ABB RobotStudio station: Simuleringsopgave_2_20200505-175028.rsstn

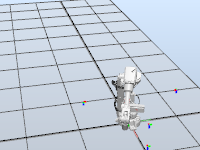
Station Simuleringsopgave_2 (saved by RobotStudio 7.0.8746.631)
Controller IRB_2600_20kg_1.65m_1
  mechanical unit ROB_1: IRB2600_20_165__02, 6 joints, base frame (0, 0, 0) mm
Layout (positions relative to the parent item):
  - IRB2600_20_165__02 [mechanism, from Robots\IRB2600_20_165_G_02.rslib] at (0, 0, 0) mm; joint values [-0.4129, 0.1779, 0.5307, -6.2924, 0.8625, 6.3308] (rad or m)
  - MyNewTool [mechanism] at (872.04, -382.72, 618.96) mm, rotated rx -179.6 ry 0 rz 153.96 deg
      TCP MyNewTool at (0, 0, 30) mm
      links: SimpleGripper
Attachment: MyNewTool is attached to IRB2600_20_165__02 / Link6
Targets, tools, work objects and paths stored in the station, written as RAPID:
! task T_ROB1
MODULE CalibData
  TASK PERS wobjdata Workobject_1:=[FALSE,TRUE,"",[[0,0,0],[1,0,0,0]],[[0,0,0],[1,0,0,0]]];
  PERS tooldata MyNewTool:=[TRUE,[[0,0,30],[1,0,0,0]],[1,[0,0,1],[1,0,0,0],0,0,0]];
ENDMODULE

! task T_ROB1
MODULE Module1
  CONST robtarget PicKUp:=[[996.139868276,-0.000086478,170.226118879],[0.000036866,0.000002225,0.999993783,-0.00352606],[0,-5,4,0],[9E+09,9E+09,9E+09,9E+09,9E+09,9E+09]];
  CONST robtarget Home:=[[996.139869233,-0.000090103,615.626718052],[0.000036871,0.000002267,0.999993783,-0.003526076],[0,-5,4,0],[9E+09,9E+09,9E+09,9E+09,9E+09,9E+09]];
  CONST robtarget Small:=[[6.065699913,-908.240962462,615.626905136],[0.002646356,-0.757323123,-0.653030822,0.002330353],[-1,-5,4,0],[9E+09,9E+09,9E+09,9E+09,9E+09,9E+09]];
  CONST robtarget Big:=[[-3.693582301,939.352796807,615.626909553],[0.002655413,-0.746102912,0.665821305,-0.002320143],[1,-5,3,0],[9E+09,9E+09,9E+09,9E+09,9E+09,9E+09]];
ENDMODULE

